# EPICS substitutions: Lakeshore340Sup/Lakeshore350.substitutions
file Lakeshore350.template {

  pattern {PORT, P, CHAN, CTRL_LOOP}
  {"\$(PORT)", "\$(P)", "A", "1"}
  {"\$(PORT)", "\$(P)", "B", "2"}
  {"\$(PORT)", "\$(P)", "C", "3"}
  {"\$(PORT)", "\$(P)", "D", "4"}
}
